FUNCTION Vector_Normalize : BOOL
VAR_IN_OUT CONSTANT
	In : Matrix;
END_VAR
VAR_IN_OUT
	Res : Matrix;
END_VAR
VAR
	Mag : LREAL;
	I : UINT;
END_VAR

IF NOT(IN.IsVector) OR NOT(Res.IsVector) OR IN.IsEmpty OR IN.Length <> Res.Length THEN
	Vector_Normalize := FALSE;
	RETURN;
END_IF

IF NOT(Vector_Magnitude(In,Res=>Mag)) THEN
	Vector_Normalize := FALSE;
	RETURN;
END_IF

//dont use copy because vectors might be in different orientations
FOR I:= 0 TO Res.Length-1 DO
	Res.SetI(I,In.GetI(I)*Mag);
END_FOR

END_FUNCTION

(* stored: Version 1.1.0.1, ProductVersion 3.1.4024.9
   POU Vector_Normalize: Id {b014a21a-b81c-08f1-053c-7e75309e191c}, SpecialFunc None *)
